Staubli VAL3: init.pgx

program init()
  local num l_nError
  local string l_sErrorMessage
begin
  //
  l_nError=mot:libLoad("Tracking\Motion")
  if l_nError!=0
    popUpMsg("Error while loading motion library: "+toString("",l_nError))
  endIf
  //
  // Start the libraries to perform conveyor tracking
  call mot:create(sConveyorList)
  //
  // Get the conveyor frame
  call mot:getConvFrame(0,fConveyor,world,l_nError)
  if l_nError!=0
    call mot:getErrorMessage(l_sErrorMessage)
    popUpMsg(l_sErrorMessage)
  endIf
  //
  // Get the detection frame
  call mot:getDetectFrame(0,fDetection,world,l_nError)
  if l_nError!=0
    call mot:getErrorMessage(l_sErrorMessage)
    popUpMsg(l_sErrorMessage)
  endIf
end
